{attribute 'qualified_only'}
{attribute 'strict'}
TYPE E_MachineState :
(
	Default := 0,
	NotHomed,
	Homing,
	Homed,
	Starting,
	Stopping,
	Running,
	StandBy,
	Error
);
END_TYPE

(* stored: Version 1.1.0.1, ProductVersion 3.1.4024.13
   DUT E_MachineState: Id {51d59891-1745-47a2-a306-168914aab215} *)
